{attribute 'qualified_only'}
{attribute 'strict'}
TYPE Permissions :
(
	User := 0, AdminUser, SuperUser
);
END_TYPE

(* stored: Version 1.1.0.1, ProductVersion 3.1.4024.4
   DUT Permissions: Id {3e44544f-024d-479c-9f7a-4f5897748ce5} *)
